# B&R Automation Studio project system-control
Automation Studio 4.5.2.102

## Configuration Config1

### Task classes (Cpu.sw)
```
Cyclic#1 (cycle 2000 us, tolerance 0 us):
  ncsdcctrl <- ncsdcctrl.prg
Cyclic#4:
  Program <- Program.prg
  Program1 <- Program1.prg
  Program2 <- Program2.prg
NcDataObjects: acp10etxen <- acp10etxen.dob, gAxis01a <- gAxis01obj.gAxis01a.dob, gAxis01i <- gAxis01obj.gAxis01i.dob, gAxis02a <- gAxis02obj.gAxis02a.dob, gAxis02i <- gAxis02obj.gAxis02i.dob, gAxis03a <- gAxis03obj.gAxis03a.dob, gAxis03i <- gAxis03obj.gAxis03i.dob, gAxis04a <- gAxis04obj.gAxis04a.dob, gAxis04i <- gAxis04obj.gAxis04i.dob
VcDataObjects: Visu <- Visu.dob
Libraries: Acp10man, Acp10par, NcGlobal, Acp10sdc, Acp10_MC, brsystem, sys_lib, runtime, AsBrStr, Library
```

### Hardware
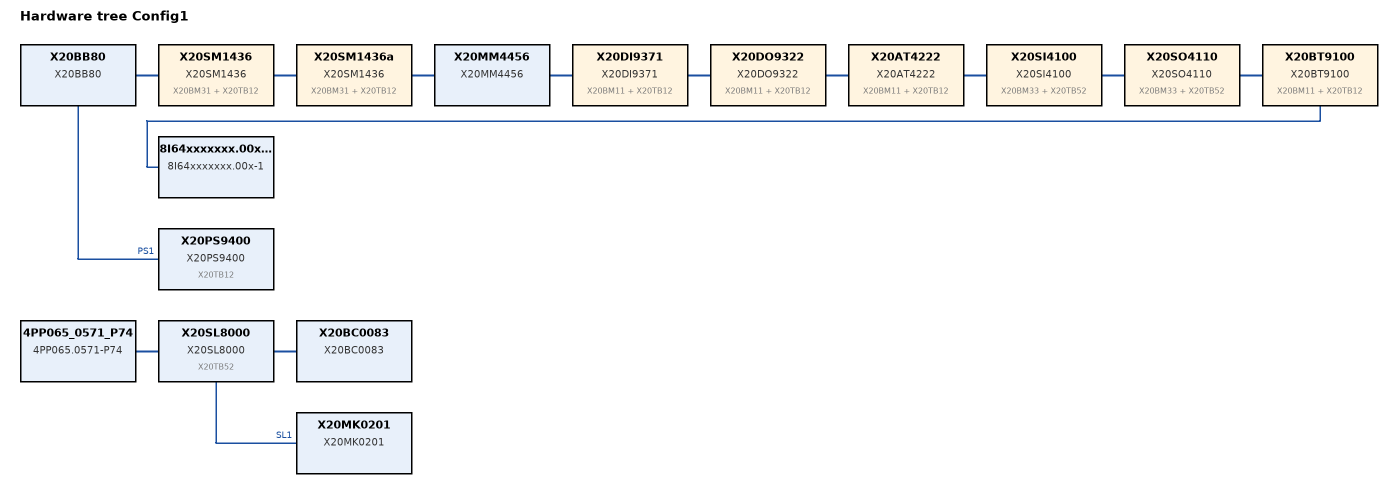
```
4PP065_0571_P74 : 4PP065.0571-P74 v1.1.2.0
  Connector IF5:
    ActivateDevice = 1
    Mode = Manual
    InternetAddress = 10.0.1.10
    SubnetMask = 255.255.255.0
    Vnc1
    VncVcObjectName1 = Visu
    VncKeyMappingFile1 = VC\PS2-Keyboard.dis
  ConfigurationID = labBR
  TimerDeviceType = EPLX2X
  TimerDevice = 4PP065_0571_P74.IF4
  TaskClassIdleTime = 2000
  Cyclic1Duration = 2000
  Cyclic1Tolerance = 0
  Cyclic1Output = 1
  VcObjectName = Visu
8I64xxxxxxx.00x-1 : 8I64xxxxxxx.00x-1 v2.1.2.0  [X2X1 -> X20BT9100.X2X1 [Cable Type=X2XCable, Length=10, Version=1.0.0.2]]
  packedETAD = packed
  packedCMDD = packed
X20AT4222 : X20AT4222 v1.2.3.0  [SS1 -> X20TB12e.SS; SL -> X20BM11b.SL1]
X20BB80 : X20BB80 v1.0.2.0
X20BC0083 : X20BC0083 v2.9.0.0  [PLK1 -> X20SL8000.PLK2 [Cable Type=PowerlinkCable, Length=10, Version=1.0.0.2]; SL -> X20BB80.SL1]
X20BM11 : X20BM11 v1.0.0.1  [X2X1 -> X20MM4456.X2X2]
X20BM11a : X20BM11 v1.0.0.1  [X2X1 -> X20BM11.X2X2]
X20BM11b : X20BM11 v1.0.0.1  [X2X1 -> X20BM11a.X2X2]
X20BM11c : X20BM11 v1.0.0.1  [X2X1 -> X20BM33a.X2X2]
X20BM31 : X20BM31 v1.0.0.1  [X2X1 -> X20BB80.IF1]
X20BM31a : X20BM31 v1.0.0.1  [X2X1 -> X20BM31.X2X2]
X20BM33 : X20BM33 v1.0.0.4  [X2X1 -> X20BM11b.X2X2]
X20BM33a : X20BM33 v1.0.0.4  [X2X1 -> X20BM33.X2X2]
X20BT9100 : X20BT9100 v1.0.3.0  [SS1 -> X20TB12f.SS; SL -> X20BM11c.SL1]
X20DI9371 : X20DI9371 v1.0.2.0  [SS1 -> X20TB12c.SS; SL -> X20BM11.SL1]
X20DO9322 : X20DO9322 v1.0.3.0  [SS1 -> X20TB12d.SS; SL -> X20BM11a.SL1]
X20MK0201 : X20MK0201 v1.0.0.0  [SL -> X20SL8000.SL1]
X20MM4456 : X20MM4456 v1.4.0.0  [X2X1 -> X20BM31a.X2X2]
X20PS9400 : X20PS9400 v1.0.2.4  [SS1 -> X20TB12.SS; PS -> X20BB80.PS1]
X20SI4100 : X20SI4100 v1.10.1.1  [SS1 -> X20TB52a.SS; SL -> X20BM33.SL1]
X20SL8000 : X20SL8000 v1.6.5.1  [PLK1 -> 4PP065_0571_P74.IF4 [Cable Type=PowerlinkCable, Length=10, Version=1.0.0.2]; PLK2 -> X20BC0083.PLK1 [Cable Type=PowerlinkCable, Length=10, Version=1.0.0.2]; SS1 -> X20TB52.SS]
  SafeProject = SafeLOGIC-1
X20SM1436 : X20SM1436 v1.4.2.1  [SS1 -> X20TB12b.SS; SL -> X20BM31.SL1]
X20SM1436a : X20SM1436 v1.4.2.1  [SS1 -> X20TB12a.SS; SL -> X20BM31a.SL1]
X20SO4110 : X20SO4110 v1.10.1.1  [SS1 -> X20TB52b.SS; SL -> X20BM33a.SL1]
  SafeModuleID = 3
X20TB12 : X20TB12 v1.0.0.0
X20TB12a : X20TB12 v1.0.0.0
X20TB12b : X20TB12 v1.0.0.0
X20TB12c : X20TB12 v1.0.0.0
X20TB12d : X20TB12 v1.0.0.0
X20TB12e : X20TB12 v1.0.0.0
X20TB12f : X20TB12 v1.0.0.0
X20TB52 : X20TB52 v1.0.0.1
X20TB52a : X20TB52 v1.0.0.1
X20TB52b : X20TB52 v1.0.0.1
```

### IoMap.iom - 4PP065_0571_P74/IoMap.iom
```iecst
VAR_CONFIG
	Cyclic#1.gAxis01_DrvIf.iLifeCnt AT %IB."X20SM1436".LifeCnt;
	Cyclic#1.gAxis01_DrvIf.iDrvOK AT %IX."X20SM1436".DrvOk01;
	Cyclic#1.gAxis01_DrvIf.oBoostCurrent AT %QX."X20SM1436".BoostCurrent01;
	Cyclic#1.gAxis01_DrvIf.oStandStillCurrent AT %QX."X20SM1436".StandstillCurrent01;
	Cyclic#1.gAxis01_DrvIf.oSetTime AT %QW."X20SM1436".SetTime01;
	Cyclic#1.gAxis01_MotorStep0 AT %QW."X20SM1436".Motor1Step0;
	Cyclic#1.gAxis01_DiDoIf.iLifeCntDriveEnable AT %IB."X20SM1436".LifeCnt;
	Cyclic#1.gAxis01_DiDoIf.iLifeCntDriveReady AT %IB."X20SM1436".LifeCnt;
	Cyclic#1.gAxis01_DiDoIf.iDriveReady AT %IX."X20SM1436".DrvOk01;
	Cyclic#1.gAxis01_DiDoIf.oDriveEnable AT %QX."X20SM1436".DriveEnable01;
	Cyclic#1.gAxis01_EncIf1.iLifeCnt AT %IB."X20SM1436".LifeCnt;
	Cyclic#1.gAxis01_EncIf1.iEncOK AT %IX."X20SM1436".EncOk01;
	Cyclic#1.gAxis01_EncIf1.iActPos AT %IW."X20SM1436".ActPos01;
	Cyclic#1.gAxis01_EncIf1.iRefPulsePos AT %IW."X20SM1436".RefPulsePos01;
	Cyclic#1.gAxis01_EncIf1.iRefPulseCnt AT %IB."X20SM1436".RefPulseCnt01;
	Cyclic#1.gAxis01_EncIf1.iActTime AT %IW."X20SM1436".ActTime01;
	Cyclic#1.gAxis02_DrvIf.iLifeCnt AT %IB."X20SM1436a".LifeCnt;
	Cyclic#1.gAxis02_DrvIf.iDrvOK AT %IX."X20SM1436a".DrvOk01;
	Cyclic#1.gAxis02_DrvIf.oBoostCurrent AT %QX."X20SM1436a".BoostCurrent01;
	Cyclic#1.gAxis02_DrvIf.oStandStillCurrent AT %QX."X20SM1436a".StandstillCurrent01;
	Cyclic#1.gAxis02_DrvIf.oSetTime AT %QW."X20SM1436a".SetTime01;
	Cyclic#1.gAxis02_MotorStep0 AT %QW."X20SM1436a".Motor1Step0;
	Cyclic#1.gAxis02_DiDoIf.iLifeCntDriveEnable AT %IB."X20SM1436a".LifeCnt;
	Cyclic#1.gAxis02_DiDoIf.iLifeCntDriveReady AT %IB."X20SM1436a".LifeCnt;
	Cyclic#1.gAxis02_DiDoIf.iDriveReady AT %IX."X20SM1436a".DrvOk01;
	Cyclic#1.gAxis02_DiDoIf.oDriveEnable AT %QX."X20SM1436a".DriveEnable01;
	Cyclic#1.gAxis02_EncIf1.iLifeCnt AT %IB."X20SM1436a".LifeCnt;
	Cyclic#1.gAxis02_EncIf1.iEncOK AT %IX."X20SM1436a".EncOk01;
	Cyclic#1.gAxis02_EncIf1.iActPos AT %IW."X20SM1436a".ActPos01;
	Cyclic#1.gAxis02_EncIf1.iRefPulsePos AT %IW."X20SM1436a".RefPulsePos01;
	Cyclic#1.gAxis02_EncIf1.iRefPulseCnt AT %IB."X20SM1436a".RefPulseCnt01;
	Cyclic#1.gAxis02_EncIf1.iActTime AT %IW."X20SM1436a".ActTime01;
	Cyclic#1.gAxis04_DrvIf.iLifeCnt AT %IB."8I64xxxxxxx.00x-1".SDC_LifeCnt;
	Cyclic#1.gAxis04_DrvIf.iDrvOK AT %IX."8I64xxxxxxx.00x-1".ETAD_Input_Bool_02;
	Cyclic#1.gAxis04_DrvIf.oSetTime AT %QW."8I64xxxxxxx.00x-1".SDC_SetTime;
	Cyclic#1.::Program:speed AT %QW."8I64xxxxxxx.00x-1".LFRD_Output;
	Cyclic#1.gAxis04_DiDoIf.iLifeCntDriveReady AT %IB."8I64xxxxxxx.00x-1".SDC_LifeCnt;
	Cyclic#1.gAxis04_DiDoIf.iLifeCntDriveEnable AT %IB."8I64xxxxxxx.00x-1".SDC_LifeCnt;
	Cyclic#1.gAxis04_DiDoIf.oDriveEnable AT %QX."8I64xxxxxxx.00x-1".CMDD_Output_Bool_00;
	Cyclic#1.gAxis04_ModuleOk AT %QX."8I64xxxxxxx.00x-1".CMDD_Output_Bool_01;
	Cyclic#1.gAxis04_ModuleOk AT %QX."8I64xxxxxxx.00x-1".CMDD_Output_Bool_02;
	Cyclic#1.gAxis04_ModuleOk AT %IX."8I64xxxxxxx.00x-1".ModuleOk;
	Cyclic#1.gAxis04_DiDoIf.oDriveEnable AT %QX."8I64xxxxxxx.00x-1".CMDD_Output_Bool_03;
	Cyclic#1.gAxis04_DiDoIf.iDriveReady AT %IX."8I64xxxxxxx.00x-1".ETAD_Input_Bool_02;
	::Program:DRIVE.STATE AT %IW."8I64xxxxxxx.00x-1".ETAD_Input;
	::Program:DRIVE.COM AT %QW."8I64xxxxxxx.00x-1".CMDD_Output;
	::led1 AT %QX."X20DO9322".DigitalOutput02;
	::led2 AT %QX."X20DO9322".DigitalOutput03;
	::led3 AT %QX."X20DO9322".DigitalOutput04;
	::led4 AT %QX."X20DO9322".DigitalOutput05;
	::Program:DRIVE.real_speed AT %IW."8I64xxxxxxx.00x-1".RFRD_Input;
END_VAR
```

## Logical view

Binary libraries used (declarations not repeated): Library

### Global.var - Global variables
```iecst
VAR
	gAxis01 : ACP10AXIS_typ;
	gAxis04 : ACP10AXIS_typ;
	gAxis02 : ACP10AXIS_typ;
	gAxis03 : ACP10AXIS_typ;
	speed_minus : INT;
	speed_plus : INT;
	ENABLED : BOOL := FALSE;
	led3 : {REDUND_UNREPLICABLE} BOOL;
	led2 : {REDUND_UNREPLICABLE} BOOL;
	led1 : {REDUND_UNREPLICABLE} BOOL;
	gAxis03_ModuleOk : BOOL := 0;
	gAxis04_ModuleOk : BOOL := 0;
	led4 : BOOL;
	gAxis01_MotorStep0 : INT := (0);
	gAxis02_MotorStep0 : INT := (0);
	gAxis01_DiDoIf : SdcDiDoIf_typ := (0);
	gAxis02_DiDoIf : SdcDiDoIf_typ := (0);
	gAxis03_DiDoIf : SdcDiDoIf_typ := (0);
	gAxis04_DiDoIf : SdcDiDoIf_typ := (0);
	gAxis04_DrvIf : SdcDrvIf16_typ := (0);
	gAxis01_DrvIf : SdcDrvIf16_typ := (0);
	gAxis03_DrvIf : SdcDrvIf16_typ := (0);
	gAxis02_DrvIf : SdcDrvIf16_typ := (0);
	gAxis02_EncIf1 : SdcEncIf16_typ := (0);
	gAxis01_EncIf1 : SdcEncIf16_typ := (0);
	gAxis02_HW : SdcHwCfg_typ := (0);
	gAxis04_HW : SdcHwCfg_typ := (0);
	gAxis01_HW : SdcHwCfg_typ := (0);
	gAxis03_HW : SdcHwCfg_typ := (0);
	Blink : BOOL;
END_VAR
```


### Program Logical/Program (ANSIC)

#### Main.c
```c
#include <bur/plctypes.h>

#ifdef _DEFAULT_INCLUDES
	#include <AsDefault.h>
#endif

void _INIT ProgramInit(void)
{
	speed=400;
	DRIVE.ENABLE=0;

}

void _CYCLIC ProgramCyclic(void)
{
	DRIVE.ENABLE = ENABLED;
	drive(&DRIVE);
}

void _EXIT ProgramExit(void)
{

}
```

### Program Logical/Program1 (ANSIC)

#### Main.c
```c
#include <bur/plctypes.h>

#ifdef _DEFAULT_INCLUDES
#include <AsDefault.h>
#endif

void _INIT ProgramInit(void)
{
	led1 = 0;
	led2 = 0;
	led3 = 0;
	led4 = 0;
}

void _CYCLIC ProgramCyclic(void)
{

	led1=LED[0];
	led2=LED[1];
	led3=LED[2];
	led4=LED[3];

}

void _EXIT ProgramExit(void)
{

}
```

- Visualisation Logical/Visu (not shown)

### Program Logical/Program2 (ANSIC)

#### Main.c
```c
#include <bur/plctypes.h>

#ifdef _DEFAULT_INCLUDES
#include <AsDefault.h>
#endif

void _INIT ProgramInit(void)
{
	led1 = 0;
	led2 = 0;
	led3 = 0;
	led4 = 0;
	Blink =0;
}

void _CYCLIC ProgramCyclic(void)
{if (Blink ==1){
		led1 = !led1;
		if(i%2){
			led2 = !led2;
		}
		if(i%7){
			led3 = !led3;
		}
		if(i%9){
			led4 = !led4;
		}
		i++;}
}

void _EXIT ProgramExit(void)
{

}
```

Listed in the project but not available here: Logical/Global.typ, Logical/ncsdcctrl, Logical/acp10etxen, Logical/gAxis01obj, Logical/gAxis02obj, Logical/gAxis03obj, Logical/gAxis04obj
